FUNCTION_BLOCK Motor
VAR_OUTPUT
	Direction: BOOL;
	Active: BOOL;
END_VAR
VAR_INPUT
	Forwards: BOOL;
	Backwards: BOOL;
	blockTime: TIME;
END_VAR
VAR
	timerForward: TOF;
	timerBackward: TOF;
	blockForward: BOOL;
	blockBackward: BOOL;
	rotateForward: BOOL;
	rotateBackward: BOOL;
	fallTrigForward: F_TRIG;
	fallDetectedForward: BOOL;
	fallTrigBackward: F_TRIG;
	fallDetectedBackward: BOOL;
END_VAR

fallTrigForward(CLK := Forwards, Q => fallDetectedForward);
fallTrigBackward(CLK := Backwards, Q => fallDetectedBackward);

timerForward(IN := fallDetectedForward, PT := blockTime, Q => blockBackward);
timerBackward(IN := fallDetectedBackward, PT := blockTime, Q => blockForward);

rotateForward := Forwards AND NOT blockForward;
rotateBackward := Backwards AND NOT blockBackward;


IF rotateForward OR rotateBackward THEN
	IF rotateForward THEN
		Direction := TRUE;
	ELSIF rotateBackward THEN 
		Direction := FALSE;
	END_IF
	
	Active := TRUE;
ELSE
	Active := FALSE;
END_IF

END_FUNCTION_BLOCK

(* stored: Version 1.1.0.1, ProductVersion 3.1.4024.12
   POU Motor: Id {13bd65e9-0070-4554-9c32-04047f08cb7f}, SpecialFunc None *)
